// Struckig
// Copyright (C) 2022 Stefan Besler

// This program is free software: you can redistribute it and/or modify
// it under the terms of the GNU General Public License as published by
// the Free Software Foundation, either version 3 of the License, or
// (at your option) any later version.

// This program is distributed in the hope that it will be useful,
// but WITHOUT ANY WARRANTY; without even the implied warranty of
// MERCHANTABILITY or FITNESS FOR A PARTICULAR PURPOSE.  See the
// GNU General Public License for more details.
//
// You should have received a copy of the GNU General Public License
// along with THIS PROGRAM.  IF NOT, see <http://www.gnu.org/licenses/>.
/// Clamps `value` to the closed interval `[minimum, maximum]`.
/// If `value` is below `minimum`, returns `minimum`.
/// If `value` is above `maximum`, returns `maximum`.
FUNCTION Clamp : LREAL
VAR_INPUT
  value : LREAL; //< Input value to clamp.
  minimum : LREAL; //< Lower bound.
  maximum : LREAL; //< Upper bound.
END_VAR

Clamp := MIN(MAX(value, minimum), maximum);

END_FUNCTION

(* stored: Version 1.1.0.1
   POU Clamp: Id {33b80c2e-f513-4ac6-8fcc-f24e2eb4571f}, SpecialFunc None *)
